// Pre-made robot messages
TYPE Message :
STRUCT CONSTANT
	Connect : STRING(30) := 'CRISTART 1 CMD Connect CRIEND';
	AliveDemo : STRING(63) := 'ALIVEJOG 40.0 50.0 40.0 30.0 30.0 0.0 0.0 0.0 0.0 CRIEND';	//Do not use, only for testing!
	EnableDemo : STRING(80) := 'CRISTART CMD';
END_STRUCT
END_TYPE

(* stored: Version 1.1.0.1, ProductVersion 3.1.4024.12
   DUT Message: Id {b3b8b37b-80bf-4447-8913-41dff30b1416} *)
